(* IEC 61131-3 sources: volt/packages/volt-lsp-iec/test-corpus/pro2193/Device/Plc Logic/Application/99 Library/Function Blocks, 12 files *)

(* ---- AttachPosToButtonFB.pou ---- *)
// Attach/detach hardware buttons when a position is activated on the HMI.
FUNCTION_BLOCK AttachPosToButtonFB
VAR_IN_OUT
	value						: PositionWithLimitsType;
END_VAR
VAR
	manualControlTrigger		: TriggerFB;
	{attribute 'no_copy'}
	Drive						: REFERENCE TO ServoDriveFB;
	attaching	: BOOL;
	counter		: INT;
	AttachTimer	: BTON;
END_VAR

%LANGUAGE ST
// Only attach hardware buttons when manual control is enabled.
manualControlTrigger.Call(CLK := value.manualActive AND SER.ManualControlEnabled);

IF manualControlTrigger.Q_Rising THEN
	attaching:=TRUE;
	counter := 0;
END_IF

IF AttachTimer.Set(attaching, 1) THEN	// Always wait a second before attaching to allow UUIDActiveScreen to have correct value
	IF hmi.UUIDActiveScreen = '' THEN
		counter := counter + 1;
	ELSE
		Drive.SetManualRefPos(value);
		HardwareButtons.F1.Attach(Drive);
		HardwareButtons.F2.Attach(Drive);
		HMI.FooterName	:= enumFooterNames.ServoDrive;	// Show correct footer
		attaching := FALSE;
	END_IF

	IF counter > 250 THEN
		attaching := FALSE;
		LogPlc.Fatal('Trying to attach an observer without a UUID');
	END_IF
END_IF

IF manualControlTrigger.Q_Falling THEN
	HardwareButtons.F1.Detach(Drive);
	HardwareButtons.F2.Detach(Drive);

	IF  HardwareButtons.F1.ObserverCount = 0
	AND HardwareButtons.F2.ObserverCount = 0
	THEN
		HMI.FooterName	:= enumFooterNames.None;
	END_IF

	Drive.Halt();
	Drive.SetManualRefPos(0);
END_IF

END_FUNCTION_BLOCK

//FB_Init is always available implicitly and it is used primarily for initialization.
//The return value is not evaluated. For a specific influence, you can also declare the
//methods explicitly and provide additional code there with the standard initialization
//code. You can evaluate the return value.
{attribute 'analysis' := '-33'}
METHOD FB_Init: BOOL
VAR_INPUT
	bInitRetains	: BOOL;							// TRUE: the retain variables are initialized (reset warm / reset cold)
	bInCopyCode		: BOOL;							// TRUE: the instance will be copied to the copy code afterward (online change)

	drive			: REFERENCE TO ServoDriveFB;
END_VAR

%LANGUAGE ST
THIS^.Drive REF= drive;

END_METHOD

(* ---- CalculateParkingPosDelayFB.pou ---- *)
// Calculate delay before Y axis starts moving towards mould. If timed perfectly, the Y axis can enter the mould just before starting to decelerate.
FUNCTION_BLOCK CalculateParkingPosDelayFB
VAR_INPUT
	xDriveMoving				: BOOL;		// Y Drive moving time is measured while high
	xMouldIsOpening				: BOOL;		// Mould starts to open (Connect to a trigger output)
	xMouldEntryAllowed			: BOOL;		// Y Drive is allowed entry into the mould
END_VAR
VAR_IN_OUT
	rMoveToParkingDelay			: REAL;		// The setting is auto-adjusted.
END_VAR
VAR_OUTPUT
	xDelayValid					: BOOL;
END_VAR
VAR
	MeasureMove					: StopwatchFB;
	udiMoveDuration				: UDINT;				// Time in ms

	Trig_MouldEntry				: TriggerFB;
	TickMouldOpenStart			: CAA.TICK;
	audiMouldOpenDuration		: ARRAY[1..5] OF UDINT;	// Time in ms
	udiLongestMouldOpenDuration	: UDINT;				// Time in ms
	i							: INT;
	diDifference				: DINT;
	udiOffset2					: UDINT;				// Time in ms. Add this constant offset to the waiting time. (for debugging)
END_VAR
VAR CONSTANT
	udiOffset					: UDINT := 20;			// Time in ms. Add this constant offset to the waiting time.
END_VAR

%LANGUAGE ST
// Calculation duration between drive move start towards waiting position, and start of deceleration
udiMoveDuration						:= MeasureMove.Monitor(in := xDriveMoving) / 1000;

// Calculate duration of moment of mould opening until the Y unit is allowed inside the mould
IF xMouldIsOpening THEN
	TickMouldOpenStart				:= TICKS.GetTick(FALSE);
END_IF

IF Trig_MouldEntry.Rising(CLK := xMouldEntryAllowed) AND TickMouldOpenStart <> 0 THEN
	udiLongestMouldOpenDuration		:= 0;
	FOR i := 1 TO 5 DO
		audiMouldOpenDuration[i]	:= SEL(i = 5, audiMouldOpenDuration[i+1], TICKU.GetElapsedTimeInUSec(TickMouldOpenStart) / 1000);
		udiLongestMouldOpenDuration	:= MAX(udiLongestMouldOpenDuration, audiMouldOpenDuration[i]);
	END_FOR
	TickMouldOpenStart				:= 0;
END_IF

{IF defined (IsSimulationMode)}
	udiLongestMouldOpenDuration		:= 2000;
{END_IF}

IF rMoveToParkingDelay > 0
AND udiMoveDuration > 0
AND udiLongestMouldOpenDuration > 0
AND SER.OperationMode <> SER_OperationModeType.SemiAuto
THEN
	xDelayValid						:= TRUE;
	diDifference					:= TO_DINT(udiLongestMouldOpenDuration - udiMoveDuration + udiOffset + udiOffset2);
	rMoveToParkingDelay				:= MAX(0, TO_REAL(diDifference) / 1000);
ELSE
	xDelayValid						:= FALSE;
END_IF

(*

Idea: calculate Y Axis movement:
measure until lrSetAccOut < 0

	pg		: L_MC1P.L_MC1P_ProfileGenerator;
	pg_par	: L_MC1P.L_MC1P_ProfileParameter;

pg_par.lrJerkAcc	:= 500000;
pg_par.lrJerkDec	:= 500000;
pg_par.lrMaxAcc		:= 50000;
pg_par.lrMaxDec		:= 50000;
pg_par.lrMaxVel		:= 5000;
pg_par.lrTargetPos	:= 2000;
pg_par.lrTargetVel	:= 0;

pg(
	scProfileParameter	:= pg_par,
	xExecute			:= ,
	xAuxExecute			:= ,
	xAbort				:= ,
	xVelMode			:= ,
	lrStartPos			:= 0,
	lrStartVel			:= 0,
	lrStartAcc			:= 0,
	xDone				=> ,
	xBusy				=> ,
	xAborted			=> ,
	xError				=> ,
	eErrorID			=> ,
	lrSetPosOut			=> ,
	lrSetVelOut			=> ,
	lrSetAccOut			=> );
*)

END_FUNCTION_BLOCK

(* ---- GetIPAddressFB.pou ---- *)
FUNCTION_BLOCK GetIPAddressFB
VAR_OUTPUT
	resultValid	: BOOL;
	currentIp	: STRING(20);
END_VAR
VAR
	execute					: BOOL := TRUE;
	ParameterRead			: L_IPAP.L_IPAP_ParameterRead;		// The L_IPAP_ParameterRead function block serves to read the device and PLC parameters of the Lenze Controller by the PLC application
	abReadBuffer			: ARRAY[1..4] OF BYTE;
END_VAR

// 0x2452:001 Active eng. port settings: IP address
// 0x2452:002 Active eng. port settings: Subnet
// 0x2452:003 Active eng. port settings: Gateway

%LANGUAGE ST
ParameterRead(
	xExecute		:= execute,
	xAbort			:= ,
	wIndex			:= 16#2452,
	bySubIndex		:= 16#1,
	udiTimeOut		:= UDINT#5000,
	pDataBuffer		:= ADR(abReadBuffer),
	udiBufferSize	:= SIZEOF(abReadBuffer),
	xDone			=> ,
	xBusy			=> ,
	xAborted		=> ,
	xError			=> ,
	eErrorId		=> ,
	udiDataRead		=> ,
	eDataType		=> );

IF  ParameterRead.xDone
AND ParameterRead.eErrorId = L_IPAP.L_IPAP_ERRORID.ERR_NoError
AND ParameterRead.eDataType = L_IPAP.L_IPAP_DATATYPE.DT_UNSIGNED_32
AND ParameterRead.udiDataRead = 4
THEN
	resultValid	:= TRUE;

	currentIp	:= CONCAT7(	TO_STRING(abReadBuffer[1]), '.',
							TO_STRING(abReadBuffer[2]), '.',
							TO_STRING(abReadBuffer[3]), '.',
							TO_STRING(abReadBuffer[4]));

ELSIF ParameterRead.xError OR ParameterRead.xAborted THEN
	resultValid	:= FALSE;
	currentIp	:= 'ERROR';
END_IF

END_FUNCTION_BLOCK

(* ---- GuardRealFB.pou ---- *)
// Guard that positions are within the limits
{attribute 'monitoring_display' := 'value.limitActive'}
FUNCTION_BLOCK GuardRealFB
VAR_IN_OUT
	value						: RealWithLimitsType;
END_VAR
VAR
	prevValue					: REAL := GVL_Constants.RealSmallest;
	PosChangeTooLargeAlarm		: SetErrorFB;
	{attribute 'no_copy'}
	moduleHandler				: L_IMHP.L_IMHP_IModuleHandler;

	manuallyUpdatePosInAutoMode	: REAL;	// Use by Brink programmers; to force change position during automatic operation of robot.
END_VAR

%LANGUAGE ST
Alarms();

// Set new position manually (also when SER is in automatic operation)
IF manuallyUpdatePosInAutoMode <> 0 THEN
	value.value					:= manuallyUpdatePosInAutoMode;
	prevValue					:= manuallyUpdatePosInAutoMode;
	manuallyUpdatePosInAutoMode	:= 0;
END_IF

// Check if new position is near the old position, prevent large changes during automatic operation
IF SER.InAutomaticOperation AND_THEN
(  prevValue > value.value + value.stepSize + 0.001
OR prevValue < value.value - value.stepSize - 0.001 )	// (add small value to account for rounding errors when comparing reals)
THEN
	PosChangeTooLargeAlarm.alarmCondition := TRUE;
	value.value := prevValue;
ELSE
	prevValue := value.value;
END_IF

END_FUNCTION_BLOCK

METHOD PRIVATE Alarms
VAR_INST
	PosTooSmallAlarm			: SetErrorFB;
	PosTooBigAlarm				: SetErrorFB;
END_VAR

%LANGUAGE ST
PosTooSmallAlarm(
	moduleHandler	:= moduleHandler,
	textRefId		:= General_Unit_Errors,
	errorId			:= 1,		// New position value was smaller than minimum.
	alarmCondition	:= value.value < value.lowerLimit,
	alarmDelay		:= 0.0,
	severity		:= enumErrorSeverity.Fault,
	reaction		:= enumErrorReaction.No_reaction,
	active			=> );

PosTooBigAlarm(
	moduleHandler	:= moduleHandler,
	textRefId		:= General_Unit_Errors,
	errorId			:= 2,		// New position value was bigger than maximum.
	alarmCondition	:= value.value > value.upperLimit,
	alarmDelay		:= 0.0,
	severity		:= enumErrorSeverity.Fault,
	reaction		:= enumErrorReaction.No_reaction,
	active			=> );

PosChangeTooLargeAlarm(
	moduleHandler	:= moduleHandler,
	textRefId		:= General_Unit_Errors,
	errorId			:= 3,		// New position value was bigger than max allowed stepsize. Position is corrected to previous value.
	alarmCondition	:= ,
	alarmDelay		:= 0.0,
	severity		:= enumErrorSeverity.Warning_Lock,
	reaction		:= enumErrorReaction.No_reaction,
	active			=> );

PosChangeTooLargeAlarm.alarmCondition	:= FALSE;
value.limitActive						:= PosTooSmallAlarm.active OR PosTooBigAlarm.active;

END_METHOD

//FB_Init is always available implicitly and it is used primarily for initialization.
//The return value is not evaluated. For a specific influence, you can also declare the
//methods explicitly and provide additional code there with the standard initialization
//code. You can evaluate the return value.
METHOD FB_Init: BOOL
VAR_INPUT
	bInitRetains	: BOOL;							// TRUE: the retain variables are initialized (reset warm / reset cold)
	bInCopyCode		: BOOL;							// TRUE: the instance will be copied to the copy code afterward (online change)

	moduleHandler	: L_IMHP.L_IMHP_IModuleHandler;
END_VAR

%LANGUAGE ST
THIS^.moduleHandler := moduleHandler;

END_METHOD

(* ---- JsonArrayFromReal.pou ---- *)
// Generate a Json array string from a series of REAL measurements.
{attribute 'no_explicit_call' := 'Do not call this FB. Only use the methods.'}
FUNCTION_BLOCK FINAL JsonArrayFromReal
EXTENDS MonitoringAddLogBase
VAR_INPUT
	jsonString			: POINTER TO STRING;
	stringSize			: UINT;
END_VAR
VAR_OUTPUT
	latestMeasurement	: REAL;
END_VAR
VAR
	// Initialize all elements in the array to some string
	measurements		: ARRAY[0..maxMeasurements] OF STRING(10) := [(maxMeasurements + 1)(arrayDefault)];
	latestIndex			: SINT(0..maxMeasurements);
END_VAR
VAR CONSTANT
	maxMeasurements		: SINT := 17;
	arrayDefault		: STRING(10) := 'y*os2# bK(';	// Random string to seed the array with
END_VAR

%LANGUAGE ST

END_FUNCTION_BLOCK

METHOD PUBLIC AddMeasurement
VAR_INPUT
	measurement		: REAL;
	roundingDigits	: USINT := 3;
END_VAR

// Bug in CODESYS!! :(
// Use this var_input:
//		roundingDigits	: USINT(0..4) := 3;
// CODESYS will throw exception on 'Generate code'
// Both of these work just fine, just not together:
//		roundingDigits	: USINT := 3;	// Ok
//		roundingDigits	: USINT(0..4);	// Ok
//		roundingDigits	: USINT(0..4) := 3;	// Exception!

%LANGUAGE ST
// Round new measurement and add to array
latestMeasurement			:= Round(measurement, roundingDigits);
measurements[latestIndex]	:= TO_STRING(latestMeasurement);

// Generate Json output string
UpdateOutputString();

// Increase index pointer for next measurement
Increment.Subrange(latestIndex, 0, maxMeasurements);

// Output data to monitoring system (optional)
CallAddLogLREAL(measurement);

END_METHOD

METHOD PRIVATE UpdateOutputString
VAR
	i				: SINT;
	length			: DINT;
END_VAR

%LANGUAGE ST
jsonString^ := '[';

FOR i := latestIndex TO 0 BY -1 DO
	// SIZEOF will return 81 for a string(80) var. Therefore stringSize - 1
	SAFECONCAT3(jsonString, measurements[i], ',', bufferSize := TO_INT(stringSize - 1));
END_FOR

IF latestIndex < maxMeasurements THEN
	FOR i := maxMeasurements TO latestIndex + 1 BY -1 DO
		IF measurements[i] = arrayDefault THEN	// Check if array element has a value already
			EXIT;
		END_IF
		SAFECONCAT3(jsonString, measurements[i], ',', TO_INT(stringSize - 1));
	END_FOR
END_IF

length	:= Stu.StrLenA(jsonString);
jsonString^[length - 1]	:= enumASCII.CLOSE_BRACKET;
jsonString^[length]		:= enumASCII.NULL;

END_METHOD

(* ---- ModuloCheckSensorOnPosition.pou ---- *)
// Check if a sensor does NOT detect a product somewhere within a window
FUNCTION_BLOCK PUBLIC ModuloCheckSensorOnPosition
VAR_INPUT
	enable					: BOOL;		// Enable the calculation
	position				: REAL;		// Actual position of C Axis
	stepDistance			: REAL;		// Step distance of C Axis
	sensorPosition			: REAL;		// Middle position of the gap where the sensor can detect something
	hysteresis				: REAL;		// Gap of the sensor measured from the sensorPosition
	sensor					: BOOL;		// Connected sensor
END_VAR
VAR_OUTPUT
	leftWindow				: BOOL;		// Trigger output: Chain just left the measuring window
	productDetected			: BOOL;		// Trigger output: A product was detected within the last window
END_VAR
VAR
	delta					: REAL;		// Result of mod function
	inWindow				: BOOL;		// Reading the sensor is enabled.
	inWindowTrigger			: TriggerFB;
	sensorDetected			: BOOL;
END_VAR

%LANGUAGE ST
IF NOT enable THEN
	leftWindow		:= FALSE;
	productDetected	:= FALSE;
	RETURN;
END_IF

// Get the remainder of position / stepDistance. This is how much the position is different.
delta				:= TO_REAL( TO_DINT(position * 10) MOD TO_DINT(stepDistance * 10) ) / 10;

// Delta goes from 0 to stepDistance. Check if sensorPosition is in range.
inWindow			:= ModuloTools.PositionReached(delta, sensorPosition, TO_DINT(stepDistance), hysteresis);

// Save result when sensor is detected within the window
sensorDetected		S= sensor AND inWindow;

// Give output when leaving window, and sensor is not detected (so a product is present).
leftWindow			:= inWindowTrigger.Falling(CLK := inWindow);
productDetected		:= leftWindow AND NOT sensorDetected;

// When leaving the window, reset result
sensorDetected		R= NOT inWindow;

END_FUNCTION_BLOCK

(* ---- MonitoringAddLogBase.pou ---- *)
{attribute 'symbol' := 'none'}
FUNCTION_BLOCK PUBLIC ABSTRACT MonitoringAddLogBase
VAR
	itfAddLog			: EdgePcLogging.IAddLog;	// Interface to AddLog method for monitoring system.
	plcDataType			: PlcDataType;				// Datatype where to output the measurement to the monitoring system too.
END_VAR

%LANGUAGE ST

END_FUNCTION_BLOCK

METHOD PROTECTED CallAddLogLINT
VAR_INPUT
	value					: LINT;  // The value to log
END_VAR

%LANGUAGE ST
// Output data to monitoring system (optional)
IF plcDataType <> 0 AND_THEN itfAddLog <> 0 AND_THEN itfAddLog.Connected THEN
	//Disable warning C0327: Implicit conversion from one enumeration type (PLCDATATYPE) to another (PLCDATATYPE (edgepclogging, x.x (brink automation)))
	{warning disable C0327}
	itfAddLog.AddLogLINT(	plcDataType := plcDataType,
							value		:= value);
	{warning restore C0327}
END_IF

END_METHOD

METHOD PROTECTED CallAddLogLREAL
VAR_INPUT
	value					: LREAL;  // The value to log
END_VAR

%LANGUAGE ST
// Output data to monitoring system (optional)
IF plcDataType <> 0 AND_THEN itfAddLog <> 0 AND_THEN itfAddLog.Connected THEN
	//Disable warning C0327: Implicit conversion from one enumeration type (PLCDATATYPE) to another (PLCDATATYPE (edgepclogging, x.x (brink automation)))
	{warning disable C0327}
	itfAddLog.AddLogLREAL(	plcDataType := plcDataType,
							value		:= value);
	{warning restore C0327}
END_IF

END_METHOD

METHOD PUBLIC SetMonitoring
VAR_INPUT
	itfAddLog		: EdgePcLogging.IAddLog;	// Optional: Interface to AddLog method for monitoring system.
	plcDataType		: PlcDataType;				// Optional: when in use, output the measurement to the monitoring system too.
END_VAR

%LANGUAGE ST
THIS^.itfAddLog		:= itfAddLog;
THIS^.plcDataType	:= plcDataType;

END_METHOD

(* ---- MouldCleaningFB.pou ---- *)
// Allows the IMM to produce a couple of shots without labels, to keep the mould clean.
{attribute 'symbol' := 'none'}
FUNCTION_BLOCK MouldCleaningFB
VAR_IN_OUT
	Data				: MouldCleaning_Data;
END_VAR
VAR//VISU
	{attribute 'symbol' := 'read'}	xActive				: BOOL;		// Mould cleaning (Shots without IML) is currently active
	{attribute 'symbol' := 'read'}	iCountDown			: INT;		// Number of shots to produce before starting mould cleaning
END_VAR
VAR
	iCleanShots			: INT;
END_VAR

%LANGUAGE ST
IF NOT Data.xEnable OR NOT PersistentVars.RecipeVars.EnableIML THEN
	iCountDown	:= Data.iInterval;
	iCleanShots	:= 0;
	xActive		:= FALSE;
END_IF

END_FUNCTION_BLOCK

// Returns true when labels should be placed in the mould
METHOD CycleWithIML : BOOL

%LANGUAGE ST
IF NOT Data.xEnable THEN
	CycleWithIML	:= TRUE;
	RETURN;
END_IF

IF NOT xActive THEN								// Mould cleaning is not activ
	iCountDown		:= iCountDown - 1;			// Count down cycles
	IF iCountDown <= 0 THEN
		iCleanShots	:= 0;
		xActive		:= TRUE;
	END_IF
ELSE
	iCleanShots		:= iCleanShots + 1;
	IF iCleanShots >= Data.iDuration THEN
		iCountDown	:= Data.iInterval;
		xActive		:= FALSE;
	END_IF
END_IF

CycleWithIML	:= NOT xActive;

END_METHOD

// Command to reset the module (Statemachine to zero state) in case of E-Stop
METHOD PUBLIC EStop : BOOL	// Returns true when drives are in standstill

%LANGUAGE ST
iCountDown	:= Data.iInterval;
iCleanShots	:= 0;
xActive		:= FALSE;
EStop		:= TRUE;

END_METHOD

(* ---- ProductionStatsFB.pou ---- *)
{attribute 'symbol' := 'none'}
FUNCTION_BLOCK ProductionStatsFB
EXTENDS SubjectProductionStatisticFB
IMPLEMENTS IAddProductionStats
VAR_INPUT
	serState					: PACK_ML.State;
END_VAR
VAR_OUTPUT
	SelectedStat				: ProductionStatsType;						// Outputs the currently selected statistic dataset to the HMI
END_VAR
VAR_IN_OUT
	StatisticsData				: ARRAY[1..NumberOfStatisticSets] OF ProductionStatsType;
END_VAR
VAR//VISU
	{attribute 'symbol' := 'readwrite'}	xResetSelectedStatistics	: BOOL;										// Reset button to reset the selected statistics
	{attribute 'symbol' := 'readwrite'}	usiStatisticsSelection		: USINT(*(1..NumberOfStatisticSets)*);		// Statistic dataset selector
	{attribute 'symbol' := 'readwrite'}	axResetStatistics			: ARRAY[1..NumberOfStatisticSets] OF BOOL;	// Reset each individual dataset
	{attribute 'symbol' := 'readwrite'}	newCavityAlias				: STRING(20);								// New alias for selected cavity
	{attribute 'symbol' := 'readwrite'}	newRejectReasonAlias		: STRING(40);								// New alias for selected reject reason
	{attribute 'symbol' := 'readwrite'}	selectedCavity				: USINT;									// Cavity selection for changing alias
	{attribute 'symbol' := 'readwrite'}	selectedRejectReason		: USINT;									// Reject reason selection for changing alias
	{attribute 'symbol' := 'readwrite'}	saveSelectedCavityAlias		: BOOL;										// Save the new alias for the selected cavity
	{attribute 'symbol' := 'readwrite'}	saveSelectedRejectReasonAlias	: BOOL;									// Save the new alias for the selected reject reason
	{attribute 'symbol' := 'read'}		strRuntime					: STRING(20);
END_VAR
VAR
	Trig_ResetSelected			: TriggerFB;
	Trig_Reset					: ARRAY[1..NumberOfStatisticSets] OF TriggerFB;
	Trig_ResetCycleStart		: TriggerFB;
	i, j						: UINT;
	k							: USINT;

	MeasureTimeStopped			: ARRAY[1..NumberOfStatisticSets] OF ONTIME;
	MeasureTimeResetting		: ARRAY[1..NumberOfStatisticSets] OF ONTIME;
	MeasureTimeIdle				: ARRAY[1..NumberOfStatisticSets] OF ONTIME;
	MeasureTimeAutomatic		: ARRAY[1..NumberOfStatisticSets] OF ONTIME;

	T_CopyToVisu				: BTON;

	debugStat					: BOOL;
	MockProduct					: ProductType;
END_VAR
VAR CONSTANT
	NumberOfStatisticSets		: USINT := 3;
END_VAR

%LANGUAGE ST
Initialize();

// Limit the selection from 1 to 3 (because VisiWinNet does not support subrange types)
usiStatisticsSelection := LIMIT(1, usiStatisticsSelection, NumberOfStatisticSets);

// Reset statistic dataset when reset button is pushed on HMI
IF Trig_ResetSelected.Falling(xResetSelectedStatistics) THEN
	Reset(usiStatisticsSelection);
END_IF

// Reset statistic dataset when reset button is pushed on HMI
FOR i := 1 TO NumberOfStatisticSets DO
	IF Trig_Reset[i].Falling(axResetStatistics[i]) THEN
		Reset(TO_USINT(i));
	END_IF
END_FOR

// Reset statistic dataset #2 when automatic cycle starts
IF Trig_ResetCycleStart.Rising(serState = PACK_ML.State.Starting) THEN
	Reset(LIMIT(1, 2, NumberOfStatisticSets));
END_IF

// Measure the On-time of the machine
FOR i := 1 TO NumberOfStatisticSets DO
	MeasureTimeStopped[i](		In := serState = PACK_ML.State.Stopped);
	MeasureTimeResetting[i](	In := serState = PACK_ML.State.Resetting);
	MeasureTimeIdle[i](			In := serState = PACK_ML.State.Idle);
	MeasureTimeAutomatic[i](	In := serState = PACK_ML.State.Execute);
END_FOR

// Copy the currently selected dataset to the HMI every second.
IF T_CopyToVisu.Set(TRUE, 1) THEN
	SelectedStat	:= StatisticsData[usiStatisticsSelection];
	T_CopyToVisu.Reset();
	FormatString();
	JsonBuilder.executeStatJson := TRUE;
END_IF

IF debugStat THEN
	Count(MockProduct);
	debugStat := FALSE;
END_IF

// Handle alias changes from visu
HandleCavityAliasChange();
HandleRejectReasonAliasChange();

END_FUNCTION_BLOCK

// Add a product to the statistics
METHOD PUBLIC Count
VAR_IN_OUT
	Product				: ProductType;
END_VAR
VAR
	xProductIsRejected	: BOOL;
	productCavityNo		: UINT;
	refStat				: REFERENCE TO ProductionStatsCavityType;
END_VAR

%LANGUAGE ST
// Check if cavity number is valid
IF Product.CavNo < GVL_Constants.CavityStartIndex
OR Product.CavNo > GVL_Constants.CavityEndIndex
OR NOT Product.Present
THEN
	RETURN;
END_IF

// Check if current product is rejected.
xProductIsRejected	:= Arrays.Bool_Any(Product.RejectReason, TRUE);

FOR i := 1 TO NumberOfStatisticSets DO

	FOR j := 1 TO 2 DO	// Do 2 loops; 1 for Totals, 1 for the current cavity number

		IF j = 1 THEN
			productCavityNo			:= 0;
			refStat					REF= StatisticsData[i].Total;					// Point reference to total production counter
		ELSE
			productCavityNo			:= Product.CavNo;
			refStat					REF= StatisticsData[i].Cavity[Product.CavNo];	// Point reference to correct cavity counter
		END_IF

		refStat.History				:= SHL(refStat.History, 1);			// Shift het history DWORD 1 plek naar links.

		Increment.AnyInt(refStat.Produced);
		IF i = 3 THEN
			NotifyData(productCavityNo, enumProductionStatsCavityType.Produced, 0, refStat.Produced);
		END_IF

		IF Product.SampleShot OR Product.UncountedReject THEN
			refStat.History.0 := FALSE;
			Increment.AnyInt(refStat.UncountedReject);
			IF i = 3 THEN
				NotifyData(productCavityNo, enumProductionStatsCavityType.UncountedReject, 0, refStat.UncountedReject);
			END_IF

		ELSIF xProductIsRejected THEN
			refStat.History.0 := TRUE;
			Increment.AnyInt(refStat.Rejected);
			IF i = 3 THEN
				NotifyData(productCavityNo, enumProductionStatsCavityType.Rejected, 0, refStat.Rejected);
			END_IF

			FOR k := 1 TO GVL_Constants.MaxRejectReasonsTotal DO
				IF Product.RejectReason[k] THEN
					Increment.AnyInt(refStat.RejectReason[k]);
					IF i = 3 THEN
						NotifyData(productCavityNo, enumProductionStatsCavityType.RejectReason, k, refStat.RejectReason[k]);
					END_IF
				END_IF
			END_FOR
		ELSE
			refStat.History.0 := FALSE;
			Increment.AnyInt(refStat.Stacked);
			IF i = 3 THEN
				NotifyData(productCavityNo, enumProductionStatsCavityType.Stacked, 0, refStat.Stacked);
			END_IF
		END_IF
	END_FOR
END_FOR

END_METHOD

// Add a product array to the statistics
METHOD PUBLIC CountArray
VAR_IN_OUT
	aProductArray		: ARRAY[*] OF ProductType;
END_VAR
VAR
	di					: DINT;
END_VAR

%LANGUAGE ST
FOR di := LOWER_BOUND(aProductArray, 1) TO UPPER_BOUND(aProductArray, 1) DO
	Count(aProductArray[di]);
END_FOR

END_METHOD

// Add a 2 dimensional product array to the statistics
METHOD PUBLIC CountArray2D
VAR_IN_OUT
	aProductArray		: ARRAY[*,*] OF ProductType;
END_VAR
VAR
	di1, di2			: DINT;
END_VAR

%LANGUAGE ST
FOR di1 := LOWER_BOUND(aProductArray, 1) TO UPPER_BOUND(aProductArray, 1) DO
	FOR di2 := LOWER_BOUND(aProductArray, 2) TO UPPER_BOUND(aProductArray, 2) DO
		Count(aProductArray[di1, di2]);
	END_FOR
END_FOR

END_METHOD

METHOD PRIVATE FormatString : BOOL
VAR
	_d		: UINT;
	_h		: Util.HOUR;
	_m		: Util.MINUTE;
	_s		: Util.SECOND;
END_VAR

%LANGUAGE ST
strRuntime		:= '';

_d			:= TO_UINT(SelectedStat.TimeAutomatic / UDINT#86400);
_h			:= TO_UINT(SelectedStat.TimeAutomatic / 3600 MOD 24);
_m			:= TO_UINT(SelectedStat.TimeAutomatic / 60 MOD 60);
_s			:= TO_UINT(SelectedStat.TimeAutomatic MOD 60);

IF _d > 0 THEN
	strRuntime		:= CONCAT3(strRuntime, TO_STRING(_d), 'd ');
END_IF

IF _h > 0 OR _d > 0 THEN
	strRuntime		:= CONCAT3(strRuntime, TO_STRING(_h), ':');
END_IF

IF _m > 0 OR _h > 0 OR _d > 0 THEN
	IF _m < 10 THEN
		strRuntime	:= CONCAT(strRuntime, '0');
	END_IF
	strRuntime		:= CONCAT3(strRuntime, TO_STRING(_m), ':');
END_IF

IF _s < 10 THEN
	strRuntime		:= CONCAT(strRuntime, '0');
END_IF
strRuntime			:= CONCAT(strRuntime, TO_STRING(_s));

END_METHOD

METHOD PRIVATE HandleCavityAliasChange : BOOL
VAR_INPUT
END_VAR

%LANGUAGE ST
IF saveSelectedCavityAlias THEN
	PersistentVars.cavityAliases[GVL_Constants.CavityStartIndex + selectedCavity] := newCavityAlias;
	JsonBuilder.executeCavityAliasJson := TRUE;
	saveSelectedCavityAlias := FALSE;
END_IF

END_METHOD

METHOD PRIVATE HandleRejectReasonAliasChange : BOOL
VAR_INPUT
END_VAR

%LANGUAGE ST
IF saveSelectedRejectReasonAlias THEN
	PersistentVars.rejectReasonDescriptions[selectedRejectReason + 1] := newRejectReasonAlias;
	JsonBuilder.executeRejectReasonAliasJson := TRUE;
	saveSelectedRejectReasonAlias := FALSE;
END_IF

END_METHOD

METHOD PROTECTED Initialize
VAR_INST
	{attribute 'init_on_onlchange' }
	initialized	: BOOL;
END_VAR

%LANGUAGE ST
IF initialized THEN
	RETURN;
END_IF

FOR i := 1 TO NumberOfStatisticSets DO
	StatisticsData[i].StatId := TO_USINT(i);		// Store the counter number in the dataset

	MeasureTimeStopped[i].SetExternalSecondsReference(		StatisticsData[i].TimeStopped);
	MeasureTimeResetting[i].SetExternalSecondsReference(	StatisticsData[i].TimeResetting);
	MeasureTimeIdle[i].SetExternalSecondsReference(			StatisticsData[i].TimeIdle);
	MeasureTimeAutomatic[i].SetExternalSecondsReference(	StatisticsData[i].TimeAutomatic);

	MeasureTimeAutomatic[i].SetExternalCyclesReference(		StatisticsData[i].AutomaticCycleStarts);
END_FOR

JsonBuilder.executeCavityAliasJson			:= TRUE;
JsonBuilder.executeRejectReasonAliasJson	:= TRUE;

initialized := TRUE;

// Warning: do not place this code in a FB_Init method!
// We are settings references here, the references are pointing to a StatisticsData[i] struct.
// This struct is an var_in_out, and this variable is not yet defined during FB_Init.

END_METHOD

METHOD PRIVATE Reset
VAR_INPUT
	usiStatIndex		: USINT(1..NumberOfStatisticSets);
END_VAR
VAR
	refStat				: REFERENCE TO ProductionStatsCavityType;
END_VAR

%LANGUAGE ST
FOR j := GVL_Constants.CavityStartIndex TO GVL_Constants.CavityEndIndex + 1 DO	// Go over all cavities, and do 1 extra loop for the totals.
	IF j > GVL_Constants.CavityEndIndex THEN
		refStat					REF= StatisticsData[usiStatIndex].Total;		// Point reference to total production counter
	ELSE
		refStat					REF= StatisticsData[usiStatIndex].Cavity[j];	// Point reference to correct cavity counter
	END_IF

	refStat.Produced			:= 0;
	refStat.Rejected			:= 0;
	refStat.UncountedReject		:= 0;
	refStat.Stacked				:= 0;
	refStat.History				:= 0;
	FOR k := 1 TO GVL_Constants.MaxRejectReasonsTotal DO
		refStat.RejectReason[k]	:= 0;
	END_FOR
END_FOR

MeasureTimeStopped[usiStatIndex].Reset();
MeasureTimeResetting[usiStatIndex].Reset();
MeasureTimeIdle[usiStatIndex].Reset();
MeasureTimeAutomatic[usiStatIndex].Reset();

END_METHOD

(* ---- ReadActualErrorFB.pou ---- *)
{attribute 'symbol' := 'none'}
FUNCTION_BLOCK ReadActualErrorFB
VAR_INPUT
	moduleHandler			: L_IMHP.L_IMHP_IModuleHandler;
END_VAR
VAR_OUTPUT
	warningActive			: BOOL;
	errorActive				: BOOL;
	requestedReaction		: enumErrorReaction;
END_VAR
VAR
	ReadActualSeverity		: L_IE1P.L_IE1P_ReadActualSeverity;
	ReadActualErrorCode		: L_IE1P.L_IE1P_ReadActualErrorCode;	// For debug
END_VAR

%LANGUAGE ST
ReadActualSeverity(
	xEnable					:= TRUE,
	ModuleHandler			:= moduleHandler,
	xDisableSubmodules		:= FALSE,
	xBusy					=> ,
	xError					=> ,
	eErrorID				=> ,
	eSeverity				=> ,
	eReaction				=> ,
	sAffectedModuleName		=> ,
	AffectedModuleHandler	=> ,
	xErrorActive			=> errorActive,
	xWarningActive			=> warningActive,
	SeverityStatus			=> ,
	ReactionStatus			=> );

CASE ReadActualSeverity.eSeverity OF
	// Drives throw errors with severity 'Fault_Qsp'.
	// Stop the automatic cycle on these kind of errors.
	L_IE1P.L_IE1P_SeverityLevel.Fault_Log,
	L_IE1P.L_IE1P_SeverityLevel.Fault_QspAppl,
	L_IE1P.L_IE1P_SeverityLevel.Fault_Qsp,
	L_IE1P.L_IE1P_SeverityLevel.Fault_Qsp_Cinh,
	L_IE1P.L_IE1P_SeverityLevel.Fault_Cinh:
		CASE ReadActualSeverity.eReaction OF
			L_IE1P.L_IE1P_Reaction.FastStop:
				requestedReaction := enumErrorReaction.FastStop;
			ELSE
				requestedReaction := enumErrorReaction.Stop;
		END_CASE
	ELSE
		CASE ReadActualSeverity.eReaction OF
			L_IE1P.L_IE1P_Reaction.No_Reaction:
				requestedReaction := enumErrorReaction.No_reaction;
			L_IE1P.L_IE1P_Reaction.NormalStop:
				requestedReaction := enumErrorReaction.Stop;
			L_IE1P.L_IE1P_Reaction.CycleStop:
				requestedReaction := enumErrorReaction.EndCycle;
			L_IE1P.L_IE1P_Reaction.FastStop:
				requestedReaction := enumErrorReaction.FastStop;
			ELSE
				ThrowException('This error reaction is not supported');
		END_CASE
END_CASE

ReadActualErrorCode(
	xEnable					:= TRUE,
	ModuleHandler			:= ReadActualSeverity.AffectedModuleHandler,
	ErrorHandler			:= ,
	xBusy					=> ,
	xError					=> ,
	eErrorID				=> ,
	xErrorActive			=> ,
	xWarningActive			=> ,
	dwErrorCode				=> ,
	eSeverity				=> );

END_FUNCTION_BLOCK

(* ---- RobotSerialNumberFB.pou ---- *)
//	This FB tries to read the serialnumber of the robot from the 'RobotSerial.txt' in the root of the SD-card.
//	Content of file is validated. The serial number should be in the format: ABC1234.
//	Where the first 3 characters are uppercase letters (A-Z) and the next 4 characters are numbers.
//	This function block uses the CAA.File library.
//	If the textfile does not exist, the FB will create the text file with the default serial number.
{attribute 'monitoring_display' := 'robotSerial'}
FUNCTION_BLOCK RobotSerialNumberFB
VAR_INPUT
	execute				: BOOL;					// Rising edge starts action; Falling edge resets outputs
	controller			: enumControllerType;	// Select type of controller (PLC)
END_VAR
VAR_OUTPUT
	busy				: BOOL;
	done				: BOOL;
	errorActive			: BOOL;
	errorDescription	: STRING(80);
	robotSerial			: STRING(7);			// The Serial number of the robot.
END_VAR
VAR
	state				: INT;
	hFile				: CAA.HANDLE;
	filePath			: STRING(80);
	readBuffer			: STRING(80);
	openFile			: FILE.Open;
	readFile			: FILE.Read;
	writeFile			: FILE.Write;
	closeFile			: FILE.Close;
	projectInfo			: ProjectInfoType;
END_VAR
VAR CONSTANT
	textFileName		: STRING(20)	:= 'RobotSerial.txt';
END_VAR

%LANGUAGE ST
CASE state OF
	// Await execute rising edge to start
	0:
		openFile(	xExecute := FALSE);
		readFile(	xExecute := FALSE);
		writeFile(	xExecute := FALSE);
		closeFile(	xExecute := FALSE);
		busy						:= FALSE;
		done						:= FALSE;
		errorActive					:= FALSE;
		errorDescription			:= '';
		hFile						:= 0;
		readBuffer					:= '';
		state						:= 10;

	10:
		IF execute THEN
			busy					:= TRUE;
			state := 100;
		END_IF

	// Check for correct controllerType setting
	100:
		CASE controller OF
			enumControllerType.Legacy32xxSeries:
				filePath			:= CONCAT('/USBStorage/', textFileName);
				Increment.AnyInt(state, 10);
			enumControllerType.C5xxSeries:
				filePath			:= CONCAT('/sdcard/', textFileName);
				Increment.AnyInt(state, 10);
			ELSE
				filePath			:= '';
				errorDescription	:= 'ControllerType is not implemented!';
				state := 400;
		END_CASE

	// Open the text file for reading
	110:
		openFile.sFileName		:= filePath;
		openFile.eFileMode		:= FILE.MODE.MREAD;
		openFile(	xExecute := TRUE);

		IF openFile.xError AND openFile.eError = FILE.ERROR.NOT_EXIST THEN	// The RobotSerial.txt file could not be found, create it.
			openFile(	xExecute := FALSE);
			state := 200;
		ELSIF openFile.xError THEN
			errorDescription	:= 'Error while opening file! See openFile.eError for details.';
			hFile				:= openFile.hFile;
			openFile(	xExecute := FALSE);
			state := 400;
		ELSIF openFile.xDone THEN
			hFile				:= openFile.hFile;
			openFile(	xExecute := FALSE);
			Increment.AnyInt(state, 10);
		END_IF

	// Read the text file contents
	120:
		readFile.hFile			:= hFile;
		readFile.udiTimeOut		:= 100000;		// 100ms Timeout
		readFile.pBuffer		:= ADR(readBuffer);
		readFile.szBuffer		:= SIZEOF(readBuffer);
		readFile(	xExecute := TRUE);

		IF readFile.xError OR readFile.xAborted THEN
			errorDescription	:= 'Error while reading the file! See readFile.eError for details.';
			readFile(	xExecute := FALSE);
			state := 400;
		ELSIF readFile.xDone THEN
			readFile(	xExecute := FALSE);
			Increment.AnyInt(state, 10);
		END_IF

	// Close the text file
	130:
		closeFile.hFile			:= hFile;
		closeFile(	xExecute := TRUE);
		IF closeFile.xError THEN
			errorDescription	:= 'Error while closing the file! See closeFile.eError for details';
			hFile				:= 0;
			closeFile(	xExecute := FALSE);
			state := 400;
		ELSIF closeFile.xDone THEN
			hFile				:= 0;
			closeFile(	xExecute := FALSE);
			Increment.AnyInt(state, 10);
		END_IF

	// Validate text file contents
	140:
		IF CheckSerialFormat(ADR(readBuffer)) THEN
			robotSerial			:= readBuffer;
			busy				:= FALSE;
			done				:= TRUE;
			state := 500;
		ELSE
			errorDescription	:= 'Serial number wrong format! Should be: SER0000 (3 letters then 4 numbers)';
			state := 400;
		END_IF

	// File is missing, try to write the file. First validate the default serial in the description field in project info
	200:
		projectInfo		:= GetProjectInfo();
		IF CheckSerialFormat(ADR(projectInfo.description)) THEN
			robotSerial			:= projectInfo.description;
			Increment.AnyInt(state, 10);
		ELSE
			errorDescription	:= 'File is missing, and not created. Project info description is invalid serial';
			state := 400;
		END_IF

	// Open the text file for writing
	210:
		openFile.sFileName		:= filePath;
		openFile.eFileMode		:= FILE.MODE.MWRITE;
		openFile(	xExecute := TRUE);
		IF openFile.xError THEN
			errorDescription	:= 'Error while opening file for writing! See openFile.eError for details.';
			hFile				:= openFile.hFile;
			openFile(	xExecute := FALSE);
			state := 400;
		ELSIF openFile.xDone THEN
			hFile				:= openFile.hFile;
			openFile(	xExecute := FALSE);
			Increment.AnyInt(state, 10);
		END_IF

	// Write the serial number
	220:
		writeFile.hFile			:= hFile;
		writeFile.udiTimeOut	:= 100000;		// 100ms Timeout
		writeFile.pBuffer		:= ADR(robotSerial);
		writeFile.szSize		:= TO_UDINT(Stu.StrLenA(pstData := ADR(robotSerial)));
		writeFile(	xExecute := TRUE);

		IF writeFile.xError OR writeFile.xAborted THEN
			errorDescription	:= 'Error while writing the file! See writeFile.eError for details.';
			writeFile(	xExecute := FALSE);
			state := 400;
		ELSIF writeFile.xDone THEN
			writeFile(	xExecute := FALSE);
			Increment.AnyInt(state, 10);
		END_IF

	// Close the text file
	230:
		closeFile.hFile			:= hFile;
		closeFile(	xExecute := TRUE);
		IF closeFile.xError THEN
			errorDescription	:= 'Error while closing the file for writing! See closeFile.eError for details';
			hFile				:= 0;
			closeFile(	xExecute := FALSE);
			state := 400;
		ELSIF closeFile.xDone THEN
			errorDescription	:= CONCAT(textFileName, ' did not exist, but was created on the SD card');
			hFile				:= 0;
			busy				:= FALSE;
			done				:= TRUE;
			closeFile(	xExecute := FALSE);
			state := 500;
		END_IF

	// Error occured - Try to close the file
	400:
		IF hFile > 0 THEN
			closeFile.hFile	:= hFile;
			closeFile(	xExecute := TRUE);
			IF closeFile.xError OR closeFile.xDone THEN
				closeFile(	xExecute := FALSE);
				hFile := 0;
			END_IF
		ELSE
			LogPlc.Error(errorDescription);
			busy				:= FALSE;
			errorActive			:= TRUE;
			state := 500;
		END_IF

	// Wait for falling edge of execute input, to reset the FB
	500:
		IF NOT execute THEN
			state := 0;
		END_IF
END_CASE

END_FUNCTION_BLOCK

METHOD PRIVATE CharIsNumber : BOOL
VAR_INPUT
	character	: BYTE;
END_VAR

%LANGUAGE ST
CharIsNumber := character >= enumASCII.NUMBER_0 AND character <= enumASCII.NUMBER_9;

END_METHOD

METHOD PRIVATE CharIsUpperCaseLetter : BOOL
VAR_INPUT
	character	: BYTE;
END_VAR

%LANGUAGE ST
CharIsUpperCaseLetter := character >= enumASCII.UPPERCASE_A AND character <= enumASCII.UPPERCASE_Z;

END_METHOD

// Validate correct robot serial number
METHOD PRIVATE CheckSerialFormat : BOOL
VAR_INPUT
	serial		: POINTER TO STRING(80);	// Input string (serial) will be changed by this method
END_VAR
VAR
	i			: SINT;
END_VAR

%LANGUAGE ST
CheckSerialFormat := FALSE;

Stu.StrTrimA(pString := serial);

IF Stu.StrLenA(pstData := serial) <> 7 THEN
	RETURN;
END_IF

Stu.StrToUpperA(pString := serial);

FOR i := 0 TO 2 DO
	IF NOT CharIsUpperCaseLetter(serial^[i]) THEN
		RETURN;
	END_IF
END_FOR

FOR i := 3 TO 6 DO
	IF NOT CharIsNumber(serial^[i]) THEN
		RETURN;
	END_IF
END_FOR

CheckSerialFormat := TRUE;

END_METHOD

(* ---- TravelDistanceFB.pou ---- *)
// Alternative for L_MC1P_MeasureDistance FB from Lenze, because we need to persist totalDistance variable
{attribute 'symbol' := 'none'}
{attribute 'monitoring_display' := 'totalDistance'}
FUNCTION_BLOCK TravelDistanceFB
VAR_INPUT
	enable			: BOOL;		// Set FALSE during homing/referencing to ignore position jumps
	actPos			: REAL;		// Current position of drive [mm]
END_VAR
VAR_IN_OUT
	totalDistance	: UDINT;	// Total accumulated distance traveled (persistent) [m]
END_VAR
VAR
	oldPos			: REAL;		// Previous position for delta calculation
	travelDistance	: REAL;
	init			: BOOL	:= TRUE;	// Flag for first execution
END_VAR

%LANGUAGE ST
IF init OR NOT enable THEN		// make sure the first cycle works correctly
	oldPos				:= actPos;
	init				:= FALSE;
	RETURN;
END_IF

// Accumulate absolute distance (bi-directional travel)
travelDistance			:= travelDistance + ABS(actPos - oldPos);

IF travelDistance >= 1000 THEN
	totalDistance		:= totalDistance + 1;
	travelDistance		:= travelDistance - 1000;
END_IF

oldPos					:= actPos;				// Store current position for next cycle

END_FUNCTION_BLOCK

// Reset total distance counter
METHOD PUBLIC Reset

%LANGUAGE ST
totalDistance		:= 0;
travelDistance		:= 0.0;
oldPos				:= actPos;

END_METHOD
